(* Logix 5000 project; controller STAT 1756-L72 rev 20.12; software revision 20.04; part 5 of 34 *)
(* tags used below, declared in another part *)
   N20 : DINT[50];
   N9 : DINT[50];
   comm : BOOL;
   DateTime : DINT[7];   // DINT array tag for retrieve wallclock time through GSV created during conversion
   ons6 : BOOL;
   op010 : DINT;
   P23 : BOOL;
   P24 : BOOL;
   real : REAL;
   S_cond_venturi : DINT;
   S_FLOW_VENTURI : DINT;
   S_Lvl_incident_bak : DINT;
   S_PH_naar_venturi : DINT;
   S_Ph_Neutral : DINT;
   S_PH_venturi : DINT;
   S_pos_V_renv : DINT;
   S_T_venturi : DINT;
   scp_bas1 : SCP;
   t1 : TIMER;
   tot_pulse_venturi : REAL;
(* BASSIN, continued *)

ROUTINE main_Bassin   (* ladder *)
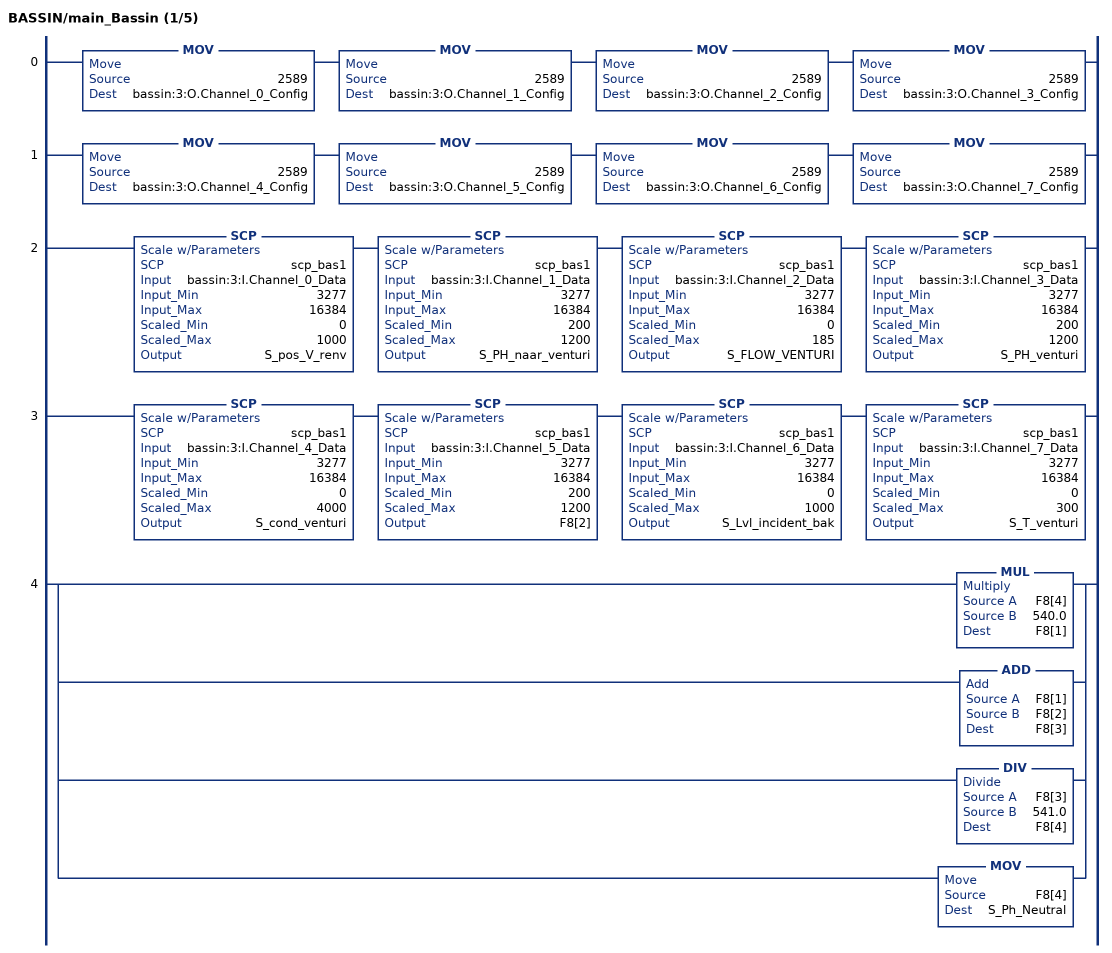
   0: MOV(2589,bassin:3:O.Channel_0_Config)MOV(2589,bassin:3:O.Channel_1_Config)MOV(2589,bassin:3:O.Channel_2_Config)MOV(2589,bassin:3:O.Channel_3_Config);
   1: MOV(2589,bassin:3:O.Channel_4_Config)MOV(2589,bassin:3:O.Channel_5_Config)MOV(2589,bassin:3:O.Channel_6_Config)MOV(2589,bassin:3:O.Channel_7_Config);
   2: SCP(scp_bas1,bassin:3:I.Channel_0_Data,3277,16384,0,1000,S_pos_V_renv)SCP(scp_bas1,bassin:3:I.Channel_1_Data,3277,16384,200,1200,S_PH_naar_venturi)SCP(scp_bas1,bassin:3:I.Channel_2_Data,3277,16384,0,185,S_FLOW_VENTURI)SCP(scp_bas1,bassin:3:I.Channel_3_Data,3277,16384,200,1200,S_PH_venturi);
   3: SCP(scp_bas1,bassin:3:I.Channel_4_Data,3277,16384,0,4000,S_cond_venturi)SCP(scp_bas1,bassin:3:I.Channel_5_Data,3277,16384,200,1200,F8[2])SCP(scp_bas1,bassin:3:I.Channel_6_Data,3277,16384,0,1000,S_Lvl_incident_bak)SCP(scp_bas1,bassin:3:I.Channel_7_Data,3277,16384,0,300,S_T_venturi);
   4: [MUL(F8[4],540.0,F8[1]) ,ADD(F8[1],F8[2],F8[3]) ,DIV(F8[3],541.0,F8[4]) ,MOV(F8[4],S_Ph_Neutral) ];
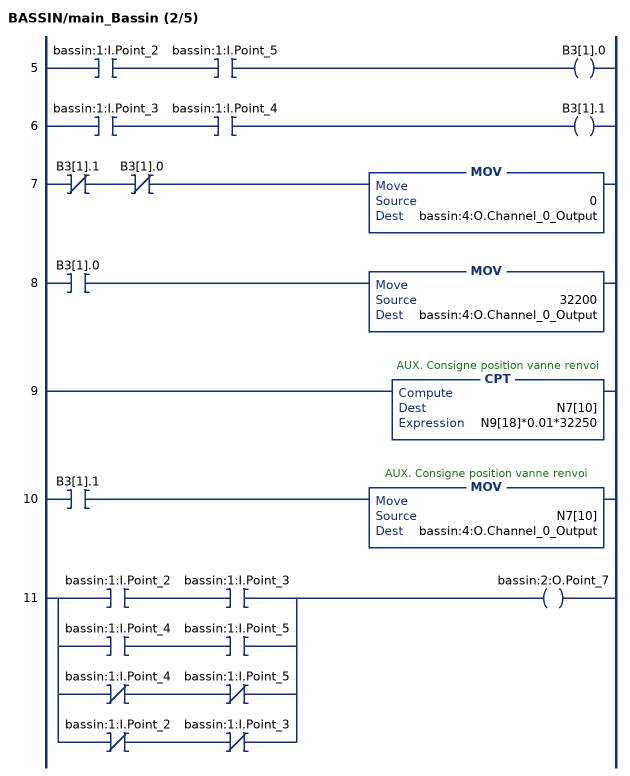
   5: XIC(bassin:1:I.Point_2)XIC(bassin:1:I.Point_5)OTE(B3[1].0);
   6: XIC(bassin:1:I.Point_3)XIC(bassin:1:I.Point_4)OTE(B3[1].1);
   7: XIO(B3[1].1)XIO(B3[1].0)MOV(0,bassin:4:O.Channel_0_Output);
   8: XIC(B3[1].0)MOV(32200,bassin:4:O.Channel_0_Output);
   9: CPT(N7[10],N9[18]*0.01*32250);
   10: XIC(B3[1].1)MOV(N7[10],bassin:4:O.Channel_0_Output);
   11: [XIC(bassin:1:I.Point_2) XIC(bassin:1:I.Point_3) ,XIC(bassin:1:I.Point_4) XIC(bassin:1:I.Point_5) ,XIO(bassin:1:I.Point_4) XIO(bassin:1:I.Point_5) ,XIO(bassin:1:I.Point_2) XIO(bassin:1:I.Point_3) ]OTE(bassin:2:O.Point_7);
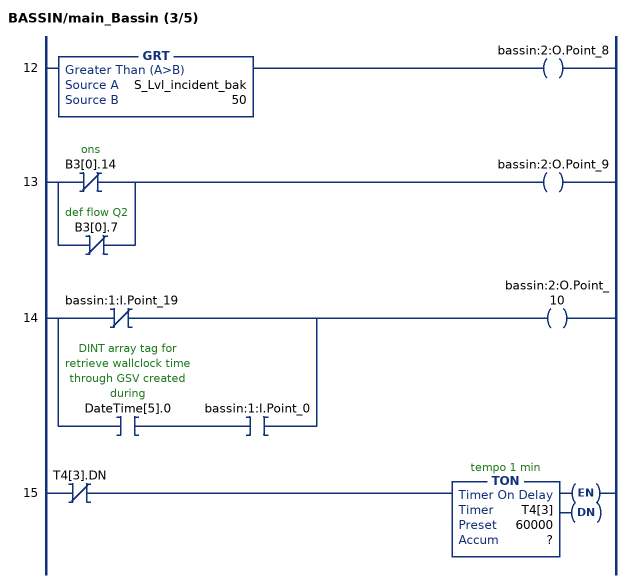
   12: GRT(S_Lvl_incident_bak,50)OTE(bassin:2:O.Point_8);
   13: [XIO(B3[0].14) ,XIO(B3[0].7) ]OTE(bassin:2:O.Point_9);
   14: [XIO(bassin:1:I.Point_19) ,XIC(DateTime[5].0) XIC(bassin:1:I.Point_0) ]OTE(bassin:2:O.Point_10);
   15: XIO(T4[3].DN)TON(T4[3],?,?);
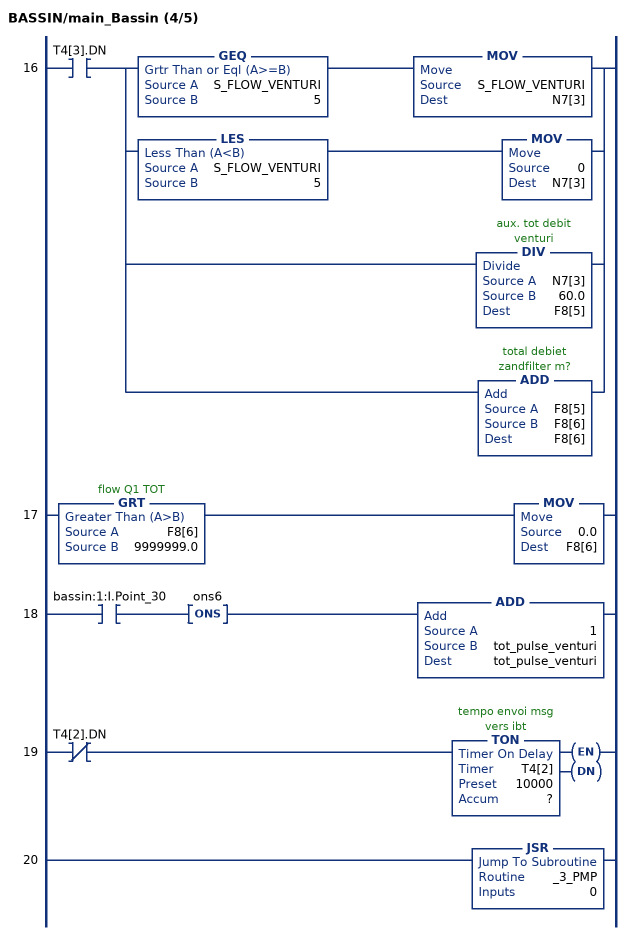
   16: XIC(T4[3].DN)[GEQ(S_FLOW_VENTURI,5) MOV(S_FLOW_VENTURI,N7[3]) ,LES(S_FLOW_VENTURI,5) MOV(0,N7[3]) ,DIV(N7[3],60.0,F8[5]) ,ADD(F8[5],F8[6],F8[6]) ];
   17: GRT(F8[6],9999999.0)MOV(0.0,F8[6]);
   18: XIC(bassin:1:I.Point_30)ONS(ons6)ADD(1,tot_pulse_venturi,tot_pulse_venturi);
   19: XIO(T4[2].DN)TON(T4[2],?,?);
   20: JSR(_3_PMP,0);
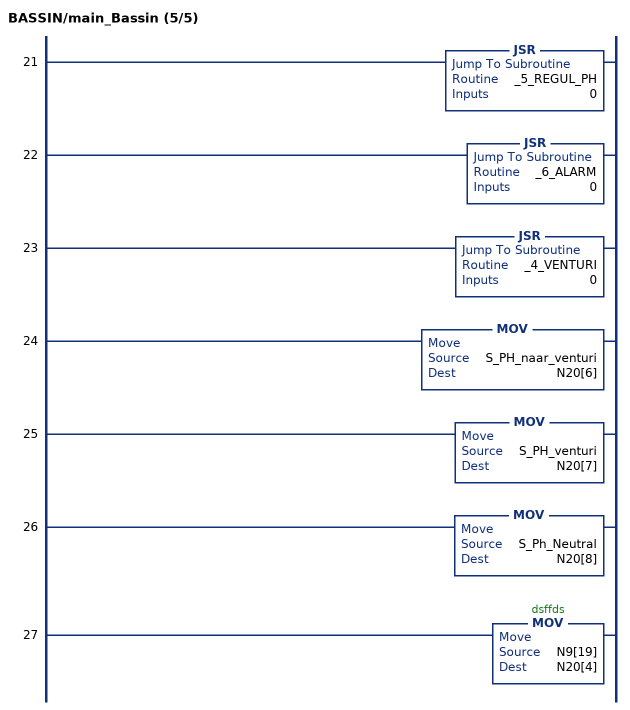
   21: JSR(_5_REGUL_PH,0);
   22: JSR(_6_ALARM,0);
   23: JSR(_4_VENTURI,0);
   24: MOV(S_PH_naar_venturi,N20[6]);
   25: MOV(S_PH_venturi,N20[7]);
   26: MOV(S_Ph_Neutral,N20[8]);
   27: MOV(N9[19],N20[4]);
END_ROUTINE
END_PROGRAM

PROGRAM ECOTECH   (* main routine ECO_Main *)
VAR
   B11 : DINT[5] := ([0] := 2#0000_0000_0000_0000_0110_0000_0000_0000, [1] := 2#0000_0000_0000_0000_1011_0000_0001_0000, [2] := 2#0000_0000_0000_0000_0000_0000_0001_0011, [3] := 2#0000_0000_0000_0000_0000_0000_0010_1000);
        [0].0   // counter pulse bit
        [0].10   // HL filter feed tank
        [0].11   // L filter feed tank
        [0].13   // OK to run backwash
        [0].14   // divert flow to filter feed tank
        [1].4   // HL water ADD off
        [1].6   // RESERVE
        [1].7   // fault filter pump
        [1].8   // RESERVE
        [1].9   // Fault APU feed pump
        [1].10   // RESERVE
        [1].11   // Fault water pump
        [1].12   // T1 not HL APU run
        [1].13   // T1 transfer stop
        [1].14   // T2 not HL APU run
        [1].15   // T2 transfer stop
        [2].0   // T3 not HL APU run
        [2].1   // T3 transfer stop
        [2].2   // T1 selected
        [2].3   // T2 selected
        [2].4   // T3 selected
        [2].8   // auto tank select
        [3].2   // monitor overide
        [3].3   // tank level OK to run
        [3].7   // unit in run mode
        [3].8   // reset
        [3].12   // alarm sound horn
   B15 : DINT[11] := ([0] := 2#0000_0000_0000_0000_0000_0000_0001_1000);
        [0].0   // RESERVE
        [0].3   // T4 not HL APU run
        [0].5   // TANK 4 MANU SELECTED
   B3 : DINT[5] := ([1] := 2#0000_0000_0000_0000_0100_1100_0001_0000, [2] := 2#0000_0000_0000_0000_0000_0000_0000_0011);
        [0].0   // PULSE_END and of cycle
        [0].2   // ARRET ENTRETIEN
        [0].5   // ons
        [0].6   // ons
        [1].0   // 0 = work by volume 1 = work by conductivity
        [1].11   // production tank level OK to run
        [1].12   // alarm condition
        [2].8   // cycle in proces
        [3].1   // backwash engeged
        [3].2   // run backwash cycle
        [3].13   // HL APU water tank
        [3].14   // LL APU water tank
        [3].15   // LL APU feed tank
        [4].0   // HL alarm APU feed tank
        [4].6   // delay between cycles
        [4].9   // end of backwash cycle
   B9 : DINT[2];
        [0].0   // aux al
   C14 : COUNTER[28] := ([27].PRE := 100);
        [0]   // RESERVE
   C5 : COUNTER[8] := ([1].PRE := 335, [2].PRE := 153, [3].PRE := 222, [4].PRE := 292, [5].PRE := 20, [5].ACC := 17, [6].PRE := 20, [7].PRE := 20, [7].ACC := 2);
        [0]   // RESERVE
        [1]   // water void volume
        [2]   // by-product volume
        [3]   // acid displ void volume valeur le 23/3/2010: 222
        [4]   // product counter valeur le 23/2/2010 292
        [5]   // T1 cycle number
        [6]   // T2 cycle number
        [7]   // T3 cycle number
   F8 : REAL[40];
        [0]   // RESERVE
   N17 : DINT[80] := ([1] := 17472, [3] := 57664, [4] := 130, [7] := 222, [8] := 292, [9] := 655, [10] := 789, [11] := 512, [12] := 808, [13] := 651, [14] := 20, [15] := 20, [16] := 20, [17] := 17, [19] := 2, [20] := 8192, [21] := 30, [22] := 1, [23] := 7, [24] := 137, [25] := 60, [28] := 5, [35] := 180, [50] := 222, [51] := 291, [54] := 621, [60] := 260, [61] := 220, [62] := 60, [63] := 292, [64] := 180, [65] := 120, [66] := 335, [67] := 153, [68] := 222, [69] := 292, [72] := 60, [74] := 456, [75] := 200, [76] := 1800, [77] := 28);
        [0]   // RESERVE
        [4].4   // flag ll l1
        [4].6   // flag ll l2
        [4].8   // flag ll l3
        [4].10   // flag ll l4
        [10]   // niveau APU feed tank
        [11]   // niveau filter feed tank
        [12]   // niveau Water APU feed Tank
        [13]   // condfuctivité 4 ma 0 mS 20 ma 300 mS
        [20]   // comm avec lancy
        [35]   // de lancy niveau op010
        [36]   // de lancy
        [37]   // de lancy
        [50]   // acid displ void volume
        [51]   // product counter
        [60]   // step 1 volume preset
        [61]   // step 2 volume preset 153 normalement
        [62]   // step 3 volume preset
        [63]   // step 4 volume preset
        [64]   // minimu vol step 1
        [65]   // min vol step2
        [66]   // step 1 volume preset old
        [67]   // step 2 volume preset old
        [68]   // step 3 volume preset old
        [69]   // step 4 volume preset old
        [70]   // volume passed in step 1
        [71]   // volume passed in step 2
        [72]   // minimum step 3 parametre
        [73]   // volume passed in step 1 + 2
        [74]   // vollmue to be reache at step 4
        [75]   // conductivity switch step 1 parametre
        [76]   // conductivity switch step 2 parametre
        [77]   // volume added on tota parametre
        [78]   // volume total
   N7 : DINT[40] := ([2] := 655, [3] := 647, [7] := 621, [9] := 28764, [20] := 48898);
        [0]   // RESERVE
        [1]   // RESERVE
        [2]   // arrivée air comprimé
        [3]   // condfuctivité 4 ma 0 mS 20 ma 300 mS
        [4]   // watervoid conductivity memo
        [5]   // by-product volume conductivity
        [6]   // acid displ void volume conductivity
        [7]   // product counter conductivity
        [18]   // DEFAUT PRIORITE 1
        [19].0   // BP ACQUIT DE SUPERVISION
        [19].1   // NEW DEFAULT
        [19].2   // NEW DEFAULT MEMO
        [20].0   // LL acid feed tank alarm light
        [20].1   // LL water feed tank alarm
        [20].2   // filter feed pump overload alarm
        [20].3   // fault filter pump
        [20].4   // overload APU feed pump alarm
        [20].5   // Fault APU feed pump
        [20].6   // overload water pump alarm
        [20].7   // Fault water pump
        [20].8   // HL T1 alarm
        [20].9   // LL alarm T1
        [20].10   // HL alarm T2
        [20].11   // LL alarm T2
        [20].12   // HL alarm T3
        [20].13   // LL alarm T3
        [20].14   // HL APU water tank
        [20].15   // LL APU water tank
        [21].0   // LL APU feed tank
        [21].1   // HL alarm APU feed tank
        [25].0   // LL acid feed tank alarm light
        [25].1   // LL water feed tank alarm
        [25].2   // filter feed pump overload alarm
        [25].3   // fault filter pump
        [25].4   // overload APU feed pump alarm
        [25].5   // Fault APU feed pump
        [25].6   // overload water pump alarm
        [25].7   // Fault water pump
        [25].8   // HL T1 alarm
        [25].9   // LL alarm T1
        [25].10   // HL alarm T2
        [25].11   // LL alarm T2
        [25].12   // HL alarm T3
        [25].13   // LL alarm T3
        [25].14   // HL APU water tank
        [25].15   // LL APU water tank
        [26].0   // LL APU feed tank
        [26].1   // HL alarm APU feed tank
        [30]   // DEFAUT EXISTANT
        [31]   // MEMO DEFAUT EXISTANT ACQUITE
        [138]   // RESERVE
        [139]   // MEMO DEFAUT DEGRAISSAGE
        [146]   // RESERVE
   R6 : CONTROL[1];
   S : INT[164] := ([0] := 16#0004, [1] := 16#0086, [2] := 16#1012, [3] := 16#a001, [4] := 16#65b3, [5] := 16#4000, [9] := 16#0003, [11] := 16#ffff, [12] := 16#ffff, [15] := 16#0b1d, [17] := 16#0002, [20] := 16#00e1, [21] := 16#0002, [22] := 16#0001, [27] := 16#ffff, [28] := 16#ffff, [33] := 16#0008, [35] := 16#0003, [37] := 16#07cb, [38] := 16#0003, [39] := 16#001c, [40] := 16#0015, [41] := 16#0015, [42] := 16#0005, [53] := 16#0004, [57] := 16#0191, [58] := 16#0001, [59] := 16#0007, [60] := 16#021e, [61] := 16#0001, [62] := 16#0003, [63] := 16#0401, [64] := 16#0023, [65] := 16#0020, [66] := 16#0200);
   T10 : TIMER[30] := ([0].PRE := 220000, [1].PRE := 220000, [2].PRE := 10000, [3].PRE := 10000, [4].PRE := 10000, [4].ACC := 10000, [4].EN := 1, [4].DN := 1, [5].PRE := 300000, [6].PRE := 300000, [7].PRE := 300000, [18].PRE := 10000, [18].ACC := 10000, [18].EN := 1, [18].DN := 1, [19].PRE := 10000, [20].PRE := 100, [21].PRE := 15000, [22].PRE := 100, [23].PRE := 15000, [24].PRE := 100, [25].PRE := 15000, [26].PRE := 20000, [27].PRE := 20000);
        [0]   // RESERVE
   T12 : TIMER[30] := ([0].PRE := 10000, [0].ACC := 10000, [0].EN := 1, [0].DN := 1, [1].PRE := 10000, [2].PRE := 10000, [3].PRE := 10000, [4].PRE := 3000, [5].PRE := 120000, [6].PRE := 10000, [10].PRE := 800, [10].ACC := 600, [10].EN := 1, [10].TT := 1, [12].PRE := 10000, [13].PRE := 10000, [14].PRE := 10000, [15].PRE := 10000, [16].PRE := 10000, [17].PRE := 10000);
        [0]   // RESERVE
   T13 : TIMER[4] := ([3].PRE := 10, [3].ACC := 11, [3].EN := 1, [3].DN := 1);
        [0]   // RESERVE
   T16 : TIMER[3] := ([1].PRE := 20000, [2].PRE := 20000);
        [0]   // RESERVE
   T4 : TIMER[30] := ([0].PRE := 10000, [1].PRE := 100, [1].ACC := 100, [3].PRE := 300000, [4].PRE := 300000, [5].PRE := 300000, [6].PRE := 312000, [7].PRE := 3000, [7].ACC := 2660, [7].EN := 1, [7].TT := 1, [13].PRE := 30000, [14].PRE := 60000, [15].PRE := 180000, [16].PRE := 150000, [17].PRE := 180000, [20].PRE := 300000, [21].PRE := 60000, [22].PRE := 10000, [23].PRE := 60000, [24].PRE := 120000, [25].PRE := 300000, [26].PRE := 2000, [27].PRE := 220000, [28].PRE := 4000, [29].PRE := 1000);
        [0]   // RESERVE
END_VAR

ROUTINE _4_PV_SUPERV   (* ladder *)
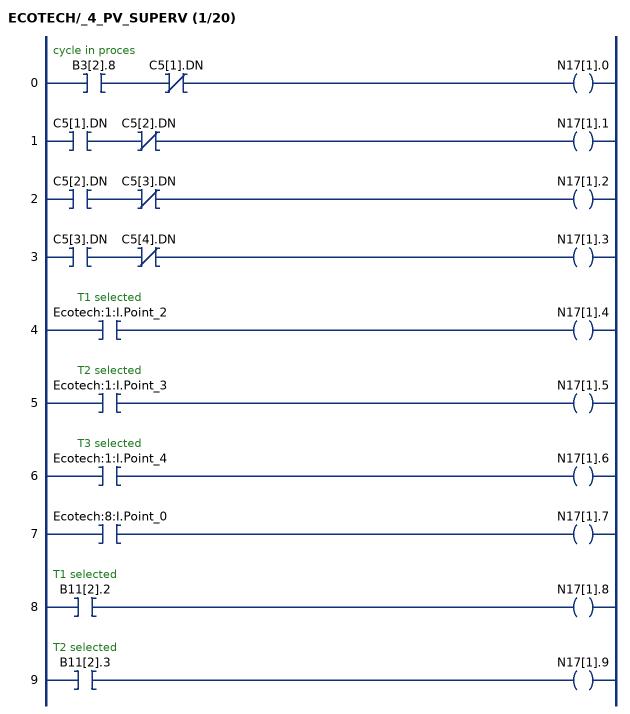
   0: XIC(B3[2].8)XIO(C5[1].DN)OTE(N17[1].0);
   1: XIC(C5[1].DN)XIO(C5[2].DN)OTE(N17[1].1);
   2: XIC(C5[2].DN)XIO(C5[3].DN)OTE(N17[1].2);
   3: XIC(C5[3].DN)XIO(C5[4].DN)OTE(N17[1].3);
   4: XIC(Ecotech:1:I.Point_2)OTE(N17[1].4);
   5: XIC(Ecotech:1:I.Point_3)OTE(N17[1].5);
   6: XIC(Ecotech:1:I.Point_4)OTE(N17[1].6);
   7: XIC(Ecotech:8:I.Point_0)OTE(N17[1].7);
   8: XIC(B11[2].2)OTE(N17[1].8);
   9: XIC(B11[2].3)OTE(N17[1].9);
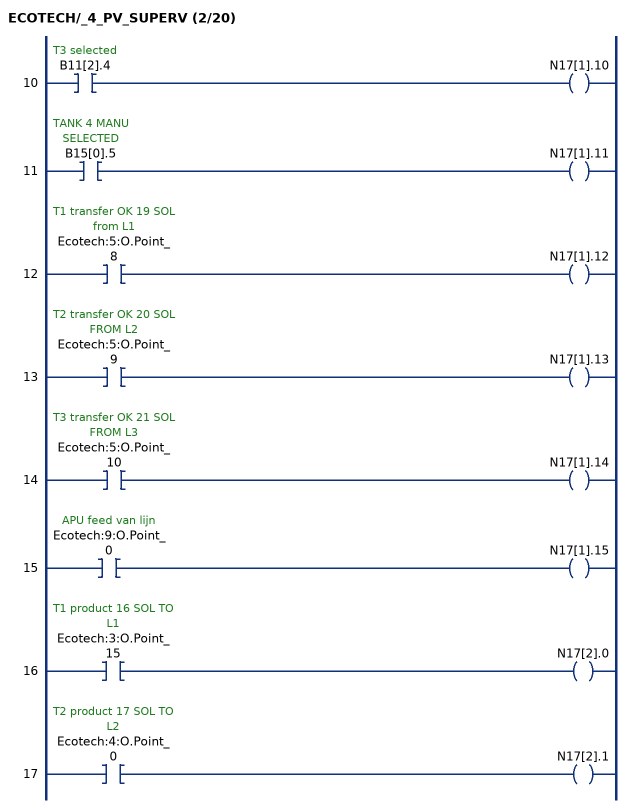
   10: XIC(B11[2].4)OTE(N17[1].10);
   11: XIC(B15[0].5)OTE(N17[1].11);
   12: XIC(Ecotech:5:O.Point_8)OTE(N17[1].12);
   13: XIC(Ecotech:5:O.Point_9)OTE(N17[1].13);
   14: XIC(Ecotech:5:O.Point_10)OTE(N17[1].14);
   15: XIC(Ecotech:9:O.Point_0)OTE(N17[1].15);
   16: XIC(Ecotech:3:O.Point_15)OTE(N17[2].0);
   17: XIC(Ecotech:4:O.Point_0)OTE(N17[2].1);
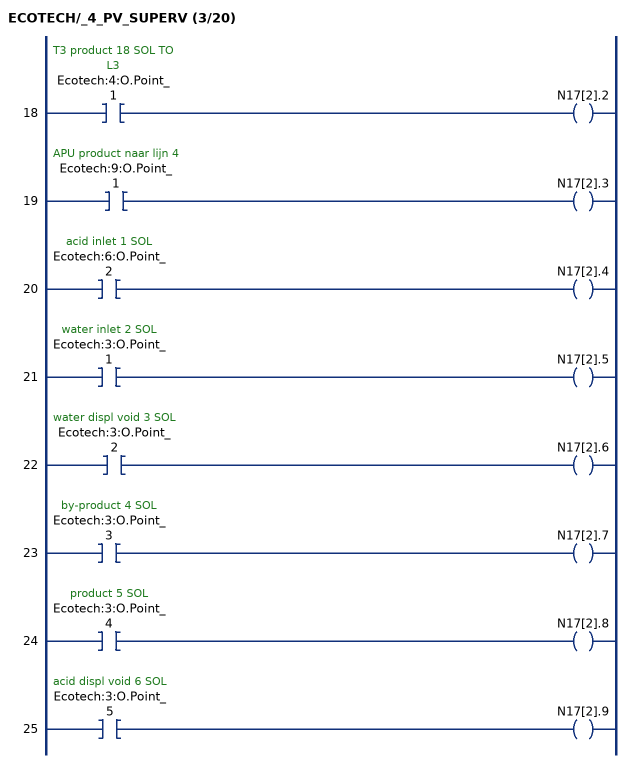
   18: XIC(Ecotech:4:O.Point_1)OTE(N17[2].2);
   19: XIC(Ecotech:9:O.Point_1)OTE(N17[2].3);
   20: XIC(Ecotech:6:O.Point_2)OTE(N17[2].4);
   21: XIC(Ecotech:3:O.Point_1)OTE(N17[2].5);
   22: XIC(Ecotech:3:O.Point_2)OTE(N17[2].6);
   23: XIC(Ecotech:3:O.Point_3)OTE(N17[2].7);
   24: XIC(Ecotech:3:O.Point_4)OTE(N17[2].8);
   25: XIC(Ecotech:3:O.Point_5)OTE(N17[2].9);
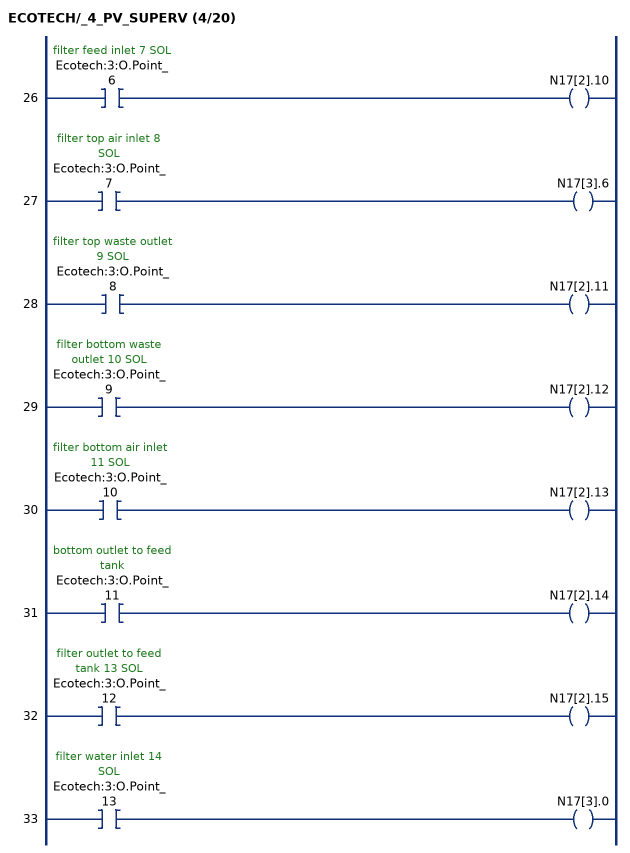
   26: XIC(Ecotech:3:O.Point_6)OTE(N17[2].10);
   27: XIC(Ecotech:3:O.Point_7)OTE(N17[3].6);
   28: XIC(Ecotech:3:O.Point_8)OTE(N17[2].11);
   29: XIC(Ecotech:3:O.Point_9)OTE(N17[2].12);
   30: XIC(Ecotech:3:O.Point_10)OTE(N17[2].13);
   31: XIC(Ecotech:3:O.Point_11)OTE(N17[2].14);
   32: XIC(Ecotech:3:O.Point_12)OTE(N17[2].15);
   33: XIC(Ecotech:3:O.Point_13)OTE(N17[3].0);
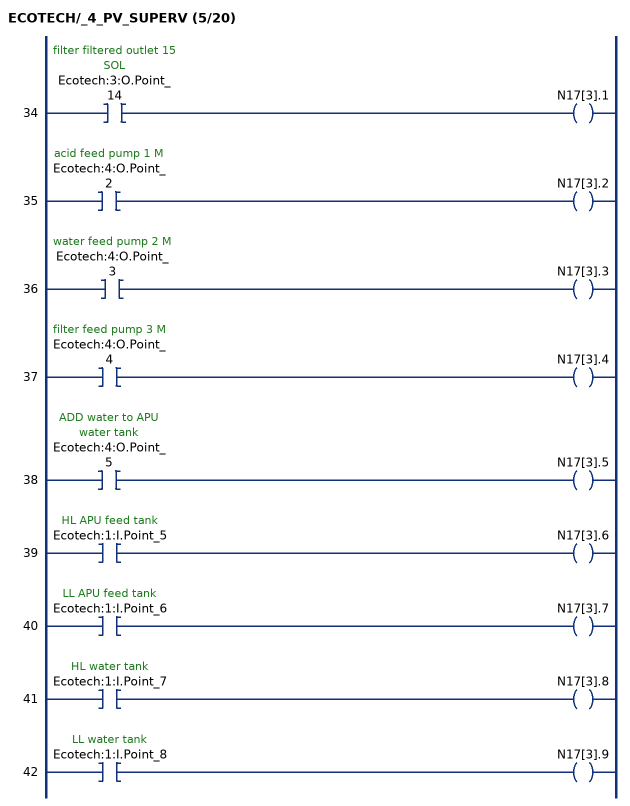
   34: XIC(Ecotech:3:O.Point_14)OTE(N17[3].1);
   35: XIC(Ecotech:4:O.Point_2)OTE(N17[3].2);
   36: XIC(Ecotech:4:O.Point_3)OTE(N17[3].3);
   37: XIC(Ecotech:4:O.Point_4)OTE(N17[3].4);
   38: XIC(Ecotech:4:O.Point_5)OTE(N17[3].5);
   39: XIC(Ecotech:1:I.Point_5)OTE(N17[3].6);
   40: XIC(Ecotech:1:I.Point_6)OTE(N17[3].7);
   41: XIC(Ecotech:1:I.Point_7)OTE(N17[3].8);
   42: XIC(Ecotech:1:I.Point_8)OTE(N17[3].9);
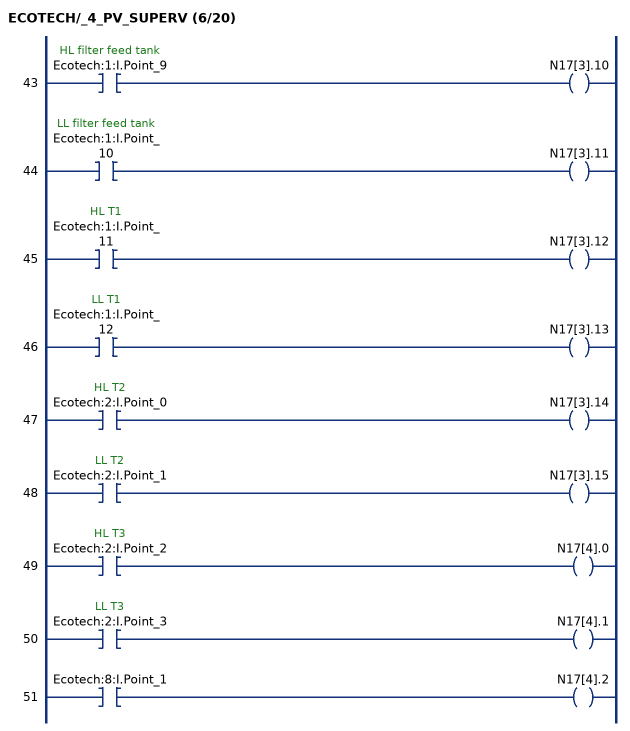
   43: XIC(Ecotech:1:I.Point_9)OTE(N17[3].10);
   44: XIC(Ecotech:1:I.Point_10)OTE(N17[3].11);
   45: XIC(Ecotech:1:I.Point_11)OTE(N17[3].12);
   46: XIC(Ecotech:1:I.Point_12)OTE(N17[3].13);
   47: XIC(Ecotech:2:I.Point_0)OTE(N17[3].14);
   48: XIC(Ecotech:2:I.Point_1)OTE(N17[3].15);
   49: XIC(Ecotech:2:I.Point_2)OTE(N17[4].0);
   50: XIC(Ecotech:2:I.Point_3)OTE(N17[4].1);
   51: XIC(Ecotech:8:I.Point_1)OTE(N17[4].2);
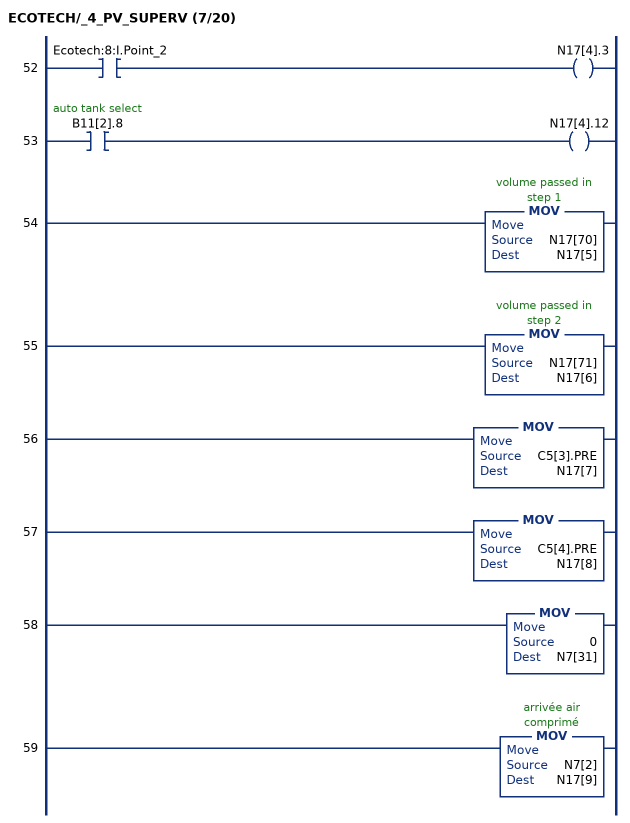
   52: XIC(Ecotech:8:I.Point_2)OTE(N17[4].3);
   53: XIC(B11[2].8)OTE(N17[4].12);
   54: MOV(N17[70],N17[5]);
   55: MOV(N17[71],N17[6]);
   56: MOV(C5[3].PRE,N17[7]);
   57: MOV(C5[4].PRE,N17[8]);
   58: MOV(0,N7[31]);
   59: MOV(N7[2],N17[9]);
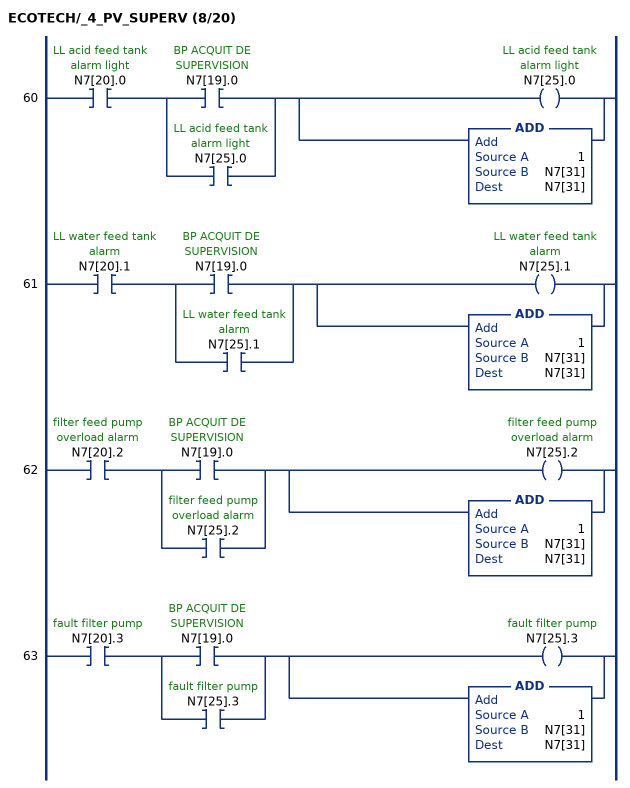
   60: XIC(N7[20].0)[XIC(N7[19].0) ,XIC(N7[25].0) ][OTE(N7[25].0) ,ADD(1,N7[31],N7[31]) ];
   61: XIC(N7[20].1)[XIC(N7[19].0) ,XIC(N7[25].1) ][OTE(N7[25].1) ,ADD(1,N7[31],N7[31]) ];
   62: XIC(N7[20].2)[XIC(N7[19].0) ,XIC(N7[25].2) ][OTE(N7[25].2) ,ADD(1,N7[31],N7[31]) ];
   63: XIC(N7[20].3)[XIC(N7[19].0) ,XIC(N7[25].3) ][OTE(N7[25].3) ,ADD(1,N7[31],N7[31]) ];
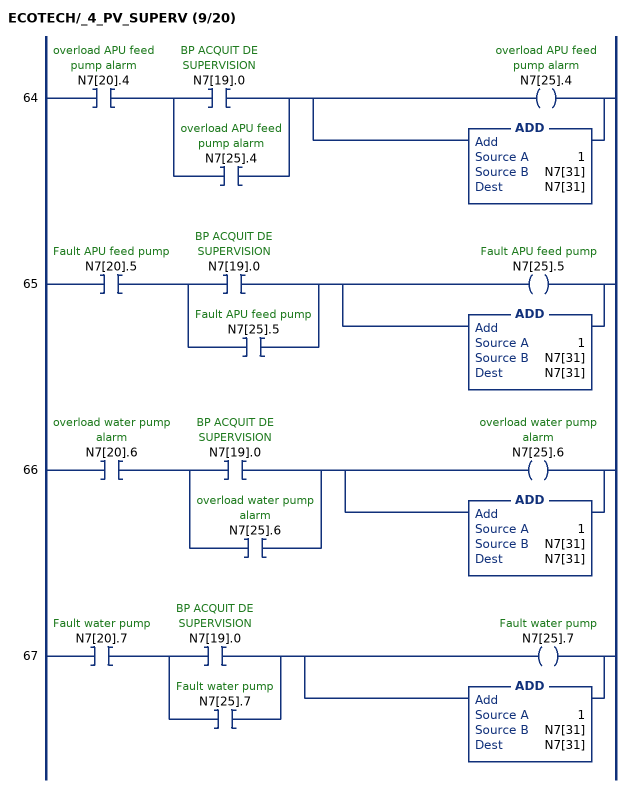
   64: XIC(N7[20].4)[XIC(N7[19].0) ,XIC(N7[25].4) ][OTE(N7[25].4) ,ADD(1,N7[31],N7[31]) ];
   65: XIC(N7[20].5)[XIC(N7[19].0) ,XIC(N7[25].5) ][OTE(N7[25].5) ,ADD(1,N7[31],N7[31]) ];
   66: XIC(N7[20].6)[XIC(N7[19].0) ,XIC(N7[25].6) ][OTE(N7[25].6) ,ADD(1,N7[31],N7[31]) ];
   67: XIC(N7[20].7)[XIC(N7[19].0) ,XIC(N7[25].7) ][OTE(N7[25].7) ,ADD(1,N7[31],N7[31]) ];
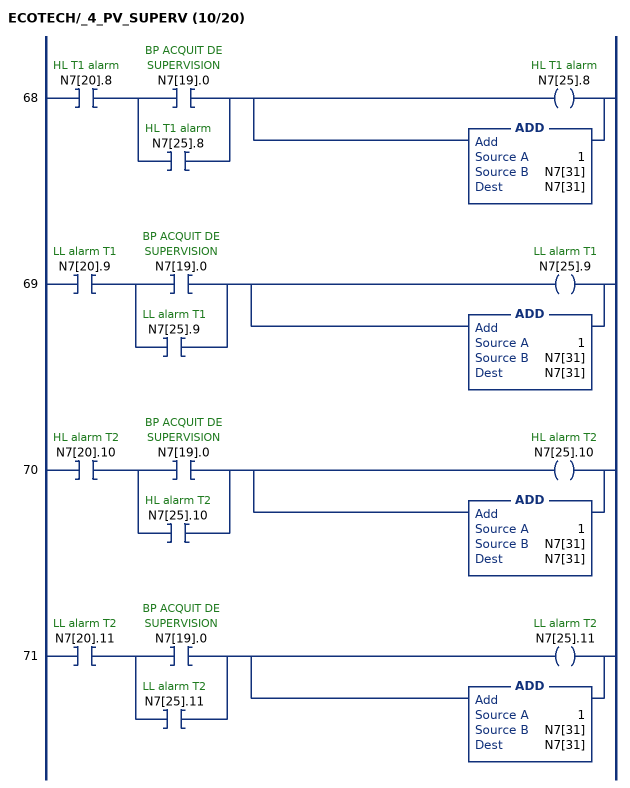
   68: XIC(N7[20].8)[XIC(N7[19].0) ,XIC(N7[25].8) ][OTE(N7[25].8) ,ADD(1,N7[31],N7[31]) ];
   69: XIC(N7[20].9)[XIC(N7[19].0) ,XIC(N7[25].9) ][OTE(N7[25].9) ,ADD(1,N7[31],N7[31]) ];
   70: XIC(N7[20].10)[XIC(N7[19].0) ,XIC(N7[25].10) ][OTE(N7[25].10) ,ADD(1,N7[31],N7[31]) ];
   71: XIC(N7[20].11)[XIC(N7[19].0) ,XIC(N7[25].11) ][OTE(N7[25].11) ,ADD(1,N7[31],N7[31]) ];
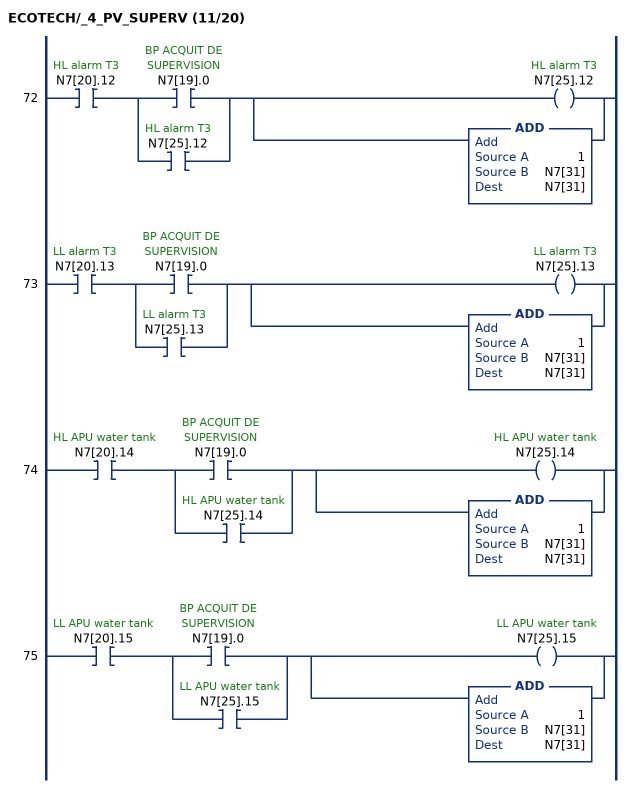
   72: XIC(N7[20].12)[XIC(N7[19].0) ,XIC(N7[25].12) ][OTE(N7[25].12) ,ADD(1,N7[31],N7[31]) ];
   73: XIC(N7[20].13)[XIC(N7[19].0) ,XIC(N7[25].13) ][OTE(N7[25].13) ,ADD(1,N7[31],N7[31]) ];
   74: XIC(N7[20].14)[XIC(N7[19].0) ,XIC(N7[25].14) ][OTE(N7[25].14) ,ADD(1,N7[31],N7[31]) ];
   75: XIC(N7[20].15)[XIC(N7[19].0) ,XIC(N7[25].15) ][OTE(N7[25].15) ,ADD(1,N7[31],N7[31]) ];
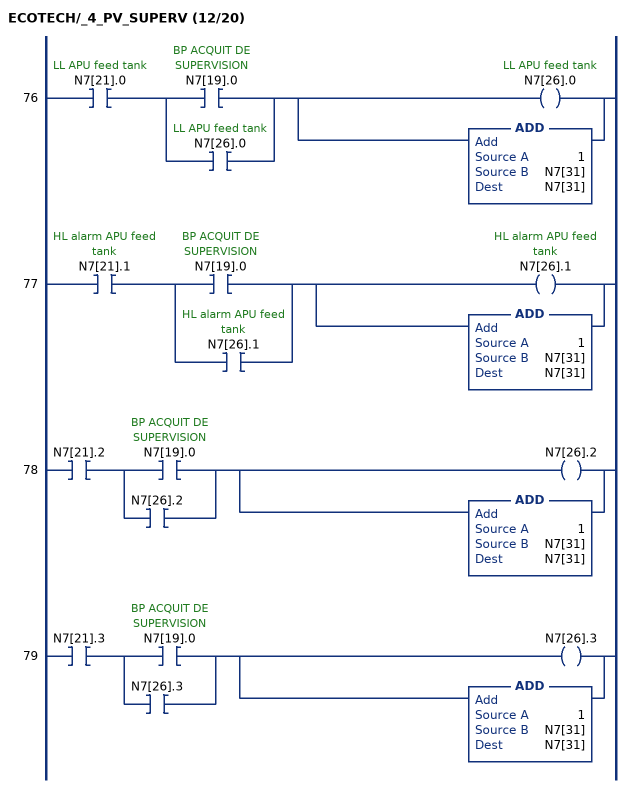
   76: XIC(N7[21].0)[XIC(N7[19].0) ,XIC(N7[26].0) ][OTE(N7[26].0) ,ADD(1,N7[31],N7[31]) ];
   77: XIC(N7[21].1)[XIC(N7[19].0) ,XIC(N7[26].1) ][OTE(N7[26].1) ,ADD(1,N7[31],N7[31]) ];
   78: XIC(N7[21].2)[XIC(N7[19].0) ,XIC(N7[26].2) ][OTE(N7[26].2) ,ADD(1,N7[31],N7[31]) ];
   79: XIC(N7[21].3)[XIC(N7[19].0) ,XIC(N7[26].3) ][OTE(N7[26].3) ,ADD(1,N7[31],N7[31]) ];
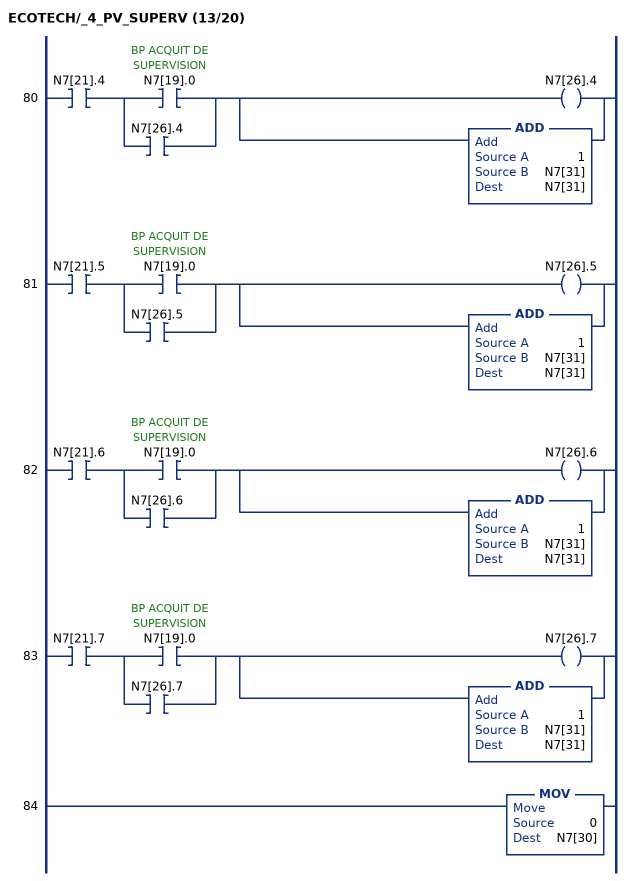
   80: XIC(N7[21].4)[XIC(N7[19].0) ,XIC(N7[26].4) ][OTE(N7[26].4) ,ADD(1,N7[31],N7[31]) ];
   81: XIC(N7[21].5)[XIC(N7[19].0) ,XIC(N7[26].5) ][OTE(N7[26].5) ,ADD(1,N7[31],N7[31]) ];
   82: XIC(N7[21].6)[XIC(N7[19].0) ,XIC(N7[26].6) ][OTE(N7[26].6) ,ADD(1,N7[31],N7[31]) ];
   83: XIC(N7[21].7)[XIC(N7[19].0) ,XIC(N7[26].7) ][OTE(N7[26].7) ,ADD(1,N7[31],N7[31]) ];
   84: MOV(0,N7[30]);
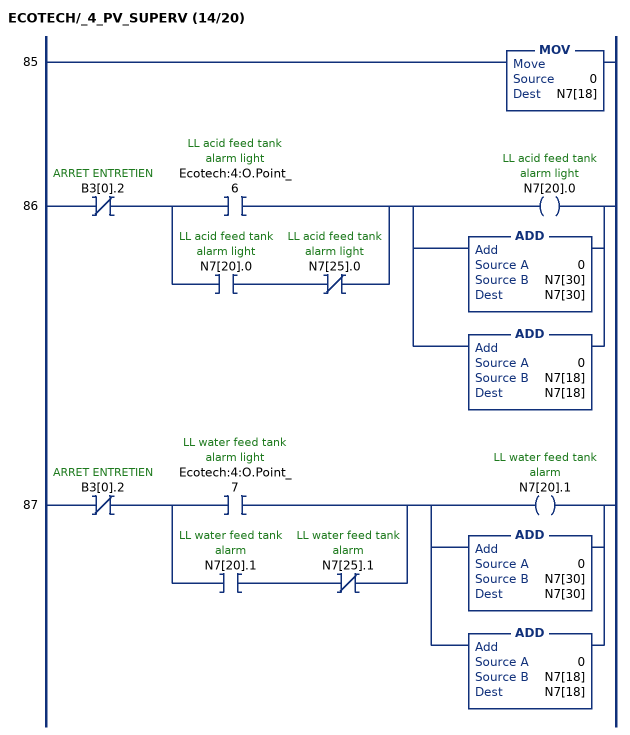
   85: MOV(0,N7[18]);
   86: XIO(B3[0].2)[XIC(Ecotech:4:O.Point_6) ,XIC(N7[20].0) XIO(N7[25].0) ][OTE(N7[20].0) ,ADD(0,N7[30],N7[30]) ,ADD(0,N7[18],N7[18]) ];
   87: XIO(B3[0].2)[XIC(Ecotech:4:O.Point_7) ,XIC(N7[20].1) XIO(N7[25].1) ][OTE(N7[20].1) ,ADD(0,N7[30],N7[30]) ,ADD(0,N7[18],N7[18]) ];
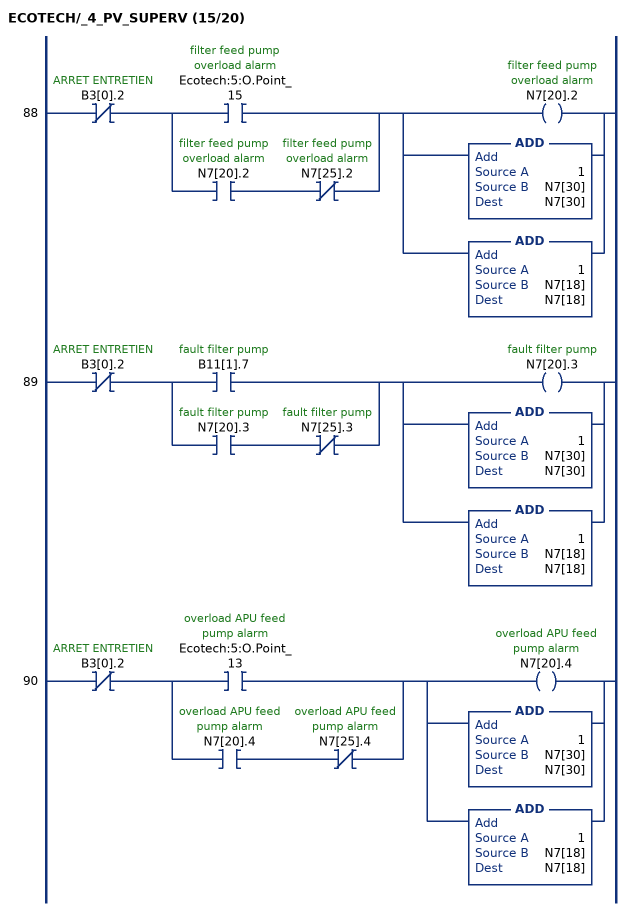
   88: XIO(B3[0].2)[XIC(Ecotech:5:O.Point_15) ,XIC(N7[20].2) XIO(N7[25].2) ][OTE(N7[20].2) ,ADD(1,N7[30],N7[30]) ,ADD(1,N7[18],N7[18]) ];
   89: XIO(B3[0].2)[XIC(B11[1].7) ,XIC(N7[20].3) XIO(N7[25].3) ][OTE(N7[20].3) ,ADD(1,N7[30],N7[30]) ,ADD(1,N7[18],N7[18]) ];
   90: XIO(B3[0].2)[XIC(Ecotech:5:O.Point_13) ,XIC(N7[20].4) XIO(N7[25].4) ][OTE(N7[20].4) ,ADD(1,N7[30],N7[30]) ,ADD(1,N7[18],N7[18]) ];
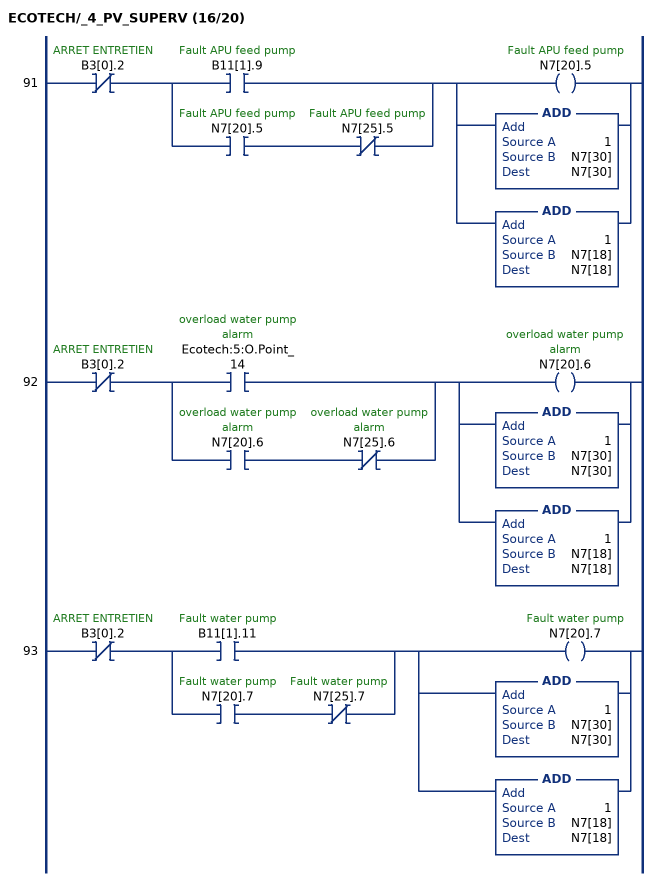
   91: XIO(B3[0].2)[XIC(B11[1].9) ,XIC(N7[20].5) XIO(N7[25].5) ][OTE(N7[20].5) ,ADD(1,N7[30],N7[30]) ,ADD(1,N7[18],N7[18]) ];
   92: XIO(B3[0].2)[XIC(Ecotech:5:O.Point_14) ,XIC(N7[20].6) XIO(N7[25].6) ][OTE(N7[20].6) ,ADD(1,N7[30],N7[30]) ,ADD(1,N7[18],N7[18]) ];
   93: XIO(B3[0].2)[XIC(B11[1].11) ,XIC(N7[20].7) XIO(N7[25].7) ][OTE(N7[20].7) ,ADD(1,N7[30],N7[30]) ,ADD(1,N7[18],N7[18]) ];
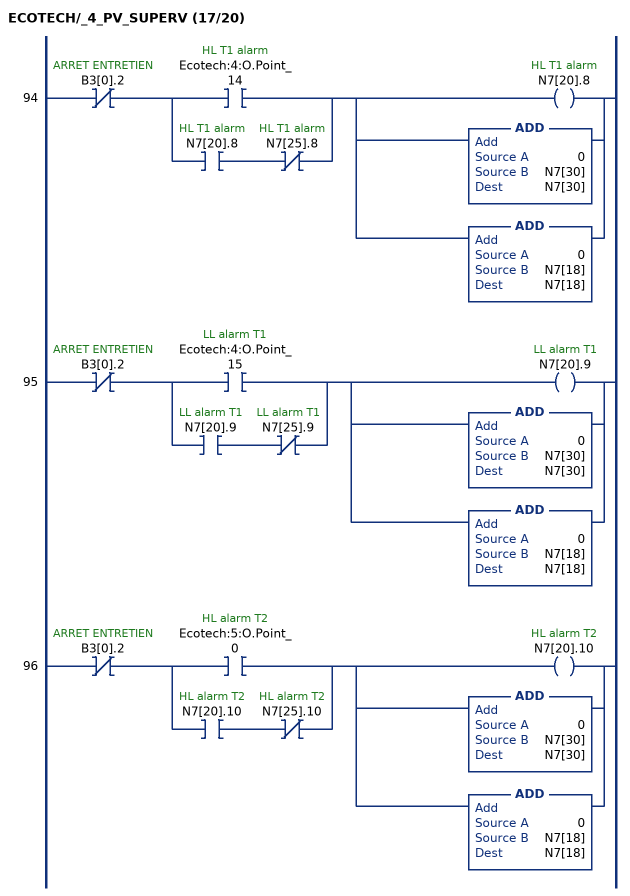
   94: XIO(B3[0].2)[XIC(Ecotech:4:O.Point_14) ,XIC(N7[20].8) XIO(N7[25].8) ][OTE(N7[20].8) ,ADD(0,N7[30],N7[30]) ,ADD(0,N7[18],N7[18]) ];
   95: XIO(B3[0].2)[XIC(Ecotech:4:O.Point_15) ,XIC(N7[20].9) XIO(N7[25].9) ][OTE(N7[20].9) ,ADD(0,N7[30],N7[30]) ,ADD(0,N7[18],N7[18]) ];
   96: XIO(B3[0].2)[XIC(Ecotech:5:O.Point_0) ,XIC(N7[20].10) XIO(N7[25].10) ][OTE(N7[20].10) ,ADD(0,N7[30],N7[30]) ,ADD(0,N7[18],N7[18]) ];
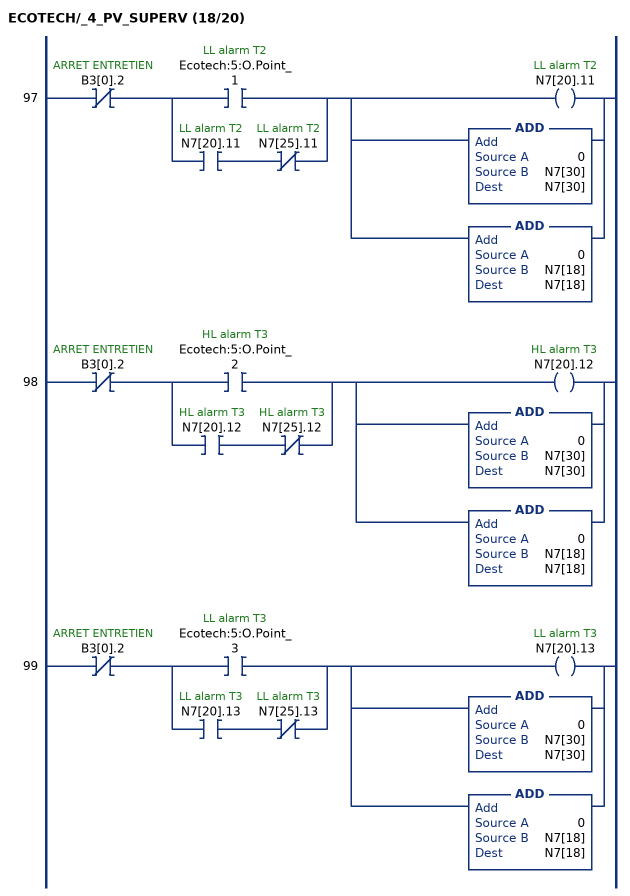
   97: XIO(B3[0].2)[XIC(Ecotech:5:O.Point_1) ,XIC(N7[20].11) XIO(N7[25].11) ][OTE(N7[20].11) ,ADD(0,N7[30],N7[30]) ,ADD(0,N7[18],N7[18]) ];
   98: XIO(B3[0].2)[XIC(Ecotech:5:O.Point_2) ,XIC(N7[20].12) XIO(N7[25].12) ][OTE(N7[20].12) ,ADD(0,N7[30],N7[30]) ,ADD(0,N7[18],N7[18]) ];
   99: XIO(B3[0].2)[XIC(Ecotech:5:O.Point_3) ,XIC(N7[20].13) XIO(N7[25].13) ][OTE(N7[20].13) ,ADD(0,N7[30],N7[30]) ,ADD(0,N7[18],N7[18]) ];
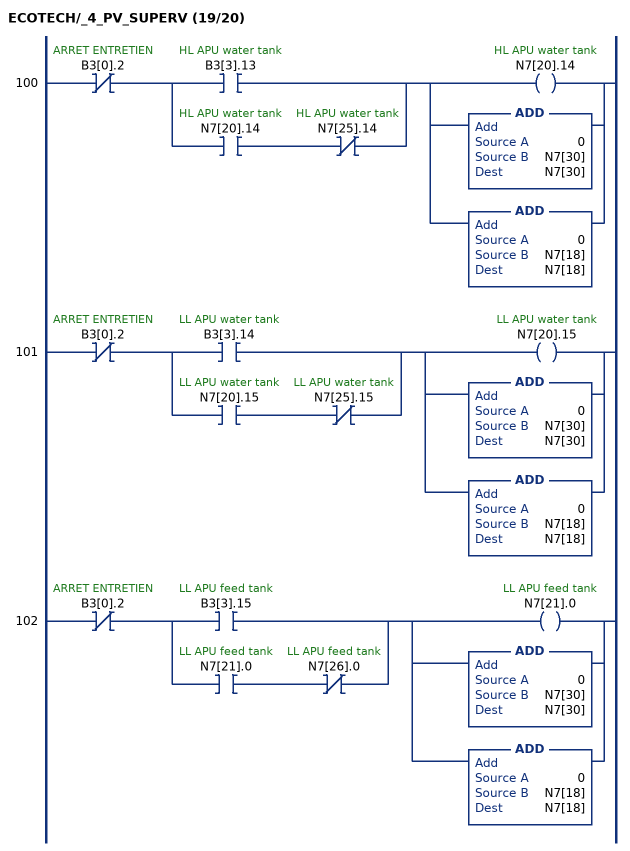
   100: XIO(B3[0].2)[XIC(B3[3].13) ,XIC(N7[20].14) XIO(N7[25].14) ][OTE(N7[20].14) ,ADD(0,N7[30],N7[30]) ,ADD(0,N7[18],N7[18]) ];
   101: XIO(B3[0].2)[XIC(B3[3].14) ,XIC(N7[20].15) XIO(N7[25].15) ][OTE(N7[20].15) ,ADD(0,N7[30],N7[30]) ,ADD(0,N7[18],N7[18]) ];
   102: XIO(B3[0].2)[XIC(B3[3].15) ,XIC(N7[21].0) XIO(N7[26].0) ][OTE(N7[21].0) ,ADD(0,N7[30],N7[30]) ,ADD(0,N7[18],N7[18]) ];
